FUNCTION F_Convert10V2Hum : INT
VAR_INPUT
	i_Value			:	INT;
END_VAR
VAR_OUTPUT
END_VAR
VAR
	r_converted2V 	: 	REAL;
	i_finalValue	:	INT;
END_VAR

// For Convertion of 0-10V Signal from 0-100%

r_converted2V := i_Value * 0.00030518509476; //Annahme 10V entspr. 32767
i_finalValue := REAL_TO_INT(r_converted2V * 10);

F_Convert10V2Hum := i_finalValue;

END_FUNCTION

(* stored: Version 1.1.0.1, ProductVersion 3.1.4024.4
   POU F_Convert10V2Hum: Id {7e32c383-4ff0-4160-8e3a-ebf080626175}, SpecialFunc None *)
